// TIA Portal V20 export
TYPE "LER_typePartDataEm6"
// stored: Access Published
   STRUCT
      stackTable : "LER_typePartData";
      stackTableBuffer : Array[0..59] of "LER_typeUnitData";
      stackTableGapVision : "LER_typeVisionGapData";
   END_STRUCT;
END_TYPE
